FUNCTION_BLOCK PUBLIC PAEEMotor2D2P EXTENDS PAEEMotorStartCtrl
VAR_INPUT
END_VAR
VAR_OUTPUT
END_VAR
VAR
	_PAPointMatInOut1 : PAPoint(THIS^);
	_PAPointMatInOut2 : PAPoint(THIS^);
	_DirectionLeft : BOOL;
	_ReqDirectionLeft : BOOL;
	_ReqSpeedFast : BOOL;
	_SpeedFast : BOOL;
	_ToggleAllowed : BOOL;
	_TransitTimeSlowFast : TIME;
END_VAR

{attribute 'monitoring' := 'call'}
//{attribute 'TcRpcEnable'}
PROPERTY PUBLIC DirectionLeft : BOOL
GET // PUBLIC
DirectionLeft := _DirectionLeft;
END_GET
SET
_DirectionLeft := DirectionLeft;
Root.OnPropertyChangedBool(THIS^, 51, _DirectionLeft);
END_SET
END_PROPERTY

METHOD FB_init : BOOL
VAR_INPUT
	bInitRetains : BOOL; // if TRUE, the retain variables are initialized (warm start / cold start)
	bInCopyCode : BOOL;  // if TRUE, the instance afterwards gets moved into the copy code (online change)
	parent : IACComponent;
END_VAR
AddPoint(_PAPointMatInOut1);
AddPoint(_PAPointMatInOut2);
END_METHOD

METHOD FB_postinit
VAR_INPUT
	root : IACVariobatch;	
END_VAR
SUPER^.FB_postinit(root);  
root.OnPropertyChangedTime(THIS^, 50, _TransitTimeSlowFast);
root.OnPropertyChangedBool(THIS^, 51, _DirectionLeft);
root.OnPropertyChangedBool(THIS^, 52, _SpeedFast);
root.OnPropertyChangedBool(THIS^, 53, _ReqDirectionLeft);
root.OnPropertyChangedBool(THIS^, 54, _ReqSpeedFast);
END_METHOD

METHOD PUBLIC HasPointReachedOffPosition : BOOL
VAR_INPUT
	point : IACPoint;
END_VAR
IF point = PAPointMatInOut1 OR point = PAPointMatInOut2 THEN
	HasPointReachedOffPosition := NOT _RunState;
ELSE
	HasPointReachedOffPosition := FALSE;
END_IF
END_METHOD

METHOD PUBLIC HasPointReachedOnPosition : BOOL
VAR_INPUT
	point : IACPoint;
END_VAR
IF point = PAPointMatInOut1 THEN
	HasPointReachedOnPosition :=	( 	(NOT _DirectionLeft) 
									 AND _RunState 
									 AND (   (_ReqSpeedFast AND _SpeedFast) 
									 	  OR (NOT _ReqSpeedFast AND NOT _SpeedFast))
									)
								OR _DirectionLeft; // Fungiert als Eingangspunkt
ELSIF point = PAPointMatInOut2 THEN
	HasPointReachedOnPosition := 	(	_DirectionLeft 
									AND _RunState 
									AND (   (_ReqSpeedFast AND _SpeedFast) 
									 	 OR (NOT _ReqSpeedFast AND NOT _SpeedFast))
									)
								OR NOT _DirectionLeft; // Fungiert als Eingangspunkt
ELSE
	HasPointReachedOnPosition := FALSE;
END_IF
END_METHOD

METHOD PUBLIC InvokeSetterBool
VAR_INPUT
	PropertyID : INT;
	PropertyValue : BOOL;
END_VAR
SUPER^.InvokeSetterBool(PropertyID, PropertyValue);
IF PropertyID = 51 THEN
	DirectionLeft := PropertyValue;
ELSIF PropertyID = 52 THEN	
	SpeedFast := PropertyValue;
ELSIF PropertyID = 53 THEN	
	ReqDirectionLeft := PropertyValue;
ELSIF PropertyID = 54 THEN	
	ReqSpeedFast := PropertyValue;
END_IF
END_METHOD

METHOD PUBLIC InvokeSetterTime
VAR_INPUT
	PropertyID : INT;
	PropertyValue : DINT;
END_VAR
SUPER^.InvokeSetterTime(PropertyID, PropertyValue);
CASE PropertyID OF
	50:
		TransitTimeSlowFast := TO_TIME(PropertyValue);
END_CASE
END_METHOD

METHOD PUBLIC IsEnabledTurnOnFastLeft : BOOL
VAR_INPUT
END_VAR
END_METHOD

METHOD PUBLIC IsEnabledTurnOnFastRight : BOOL
VAR_INPUT
END_VAR
END_METHOD

METHOD PUBLIC IsEnabledTurnOnSlowLeft : BOOL
VAR_INPUT
END_VAR
END_METHOD

METHOD PUBLIC IsEnabledTurnOnSlowRight : BOOL
VAR_INPUT
END_VAR
END_METHOD

METHOD OnInitMemory
VAR_INPUT
	root : IACVariobatch;
END_VAR
RegisterProperty(root, 50, GCL.cSizeTIME); //TransitTimeSlowFast
RegisterProperty(root, 51, GCL.cSizeBYTE); //DirectionLeft
RegisterProperty(root, 52, GCL.cSizeBYTE); //SpeedFast
RegisterProperty(root, 53, GCL.cSizeBYTE); //ReqDirectionLeft
RegisterProperty(root, 54, GCL.cSizeBYTE); //ReqSpeedFast
SUPER^.OnInitMemory(root);
END_METHOD

PROPERTY PUBLIC PAPointMatInOut1 : IACPoint
GET
PAPointMatInOut1 := _PAPointMatInOut1;
END_GET
END_PROPERTY

PROPERTY PUBLIC PAPointMatInOut2 : IACPoint
GET // PUBLIC
PAPointMatInOut2 := _PAPointMatInOut2;
END_GET
END_PROPERTY

{attribute 'monitoring' := 'call'}
//{attribute 'TcRpcEnable'}
PROPERTY PUBLIC ReqDirectionLeft : BOOL
GET // PUBLIC
ReqDirectionLeft := _ReqDirectionLeft;
END_GET
SET // PUBLIC
_ReqDirectionLeft := ReqDirectionLeft;
Root.OnPropertyChangedBool(THIS^, 53, _ReqDirectionLeft);
IF Root.InSimulation THEN
	DirectionLeft := _ReqDirectionLeft;
END_IF
END_SET
END_PROPERTY

{attribute 'monitoring' := 'call'}
//{attribute 'TcRpcEnable'}
PROPERTY PUBLIC ReqSpeedFast : BOOL
GET // PUBLIC
ReqSpeedFast := _ReqSpeedFast;
END_GET
SET // PUBLIC
_ReqSpeedFast := ReqSpeedFast;
Root.OnPropertyChangedBool(THIS^, 54, _ReqSpeedFast);
IF Root.InSimulation THEN
	SpeedFast := _ReqSpeedFast;
END_IF
END_SET
END_PROPERTY

{attribute 'monitoring' := 'call'}
//{attribute 'TcRpcEnable'}
PROPERTY PUBLIC SpeedFast : BOOL
GET
SpeedFast := _SpeedFast;
END_GET
SET // PUBLIC
_SpeedFast := SpeedFast;
Root.OnPropertyChangedBool(THIS^, 52, _SpeedFast);
END_SET
END_PROPERTY

{attribute 'monitoring' := 'call'}
//{attribute 'TcRpcEnable'}
PROPERTY PUBLIC ToggleAllowed : BOOL
GET // PUBLIC
ToggleAllowed := _ToggleAllowed;
END_GET
SET // PUBLIC
_ToggleAllowed := ToggleAllowed;
END_SET
END_PROPERTY

{attribute 'monitoring' := 'call'}
//{attribute 'TcRpcEnable'}
PROPERTY PUBLIC TransitTimeSlowFast : TIME
GET // PUBLIC
TransitTimeSlowFast := _TransitTimeSlowFast;
END_GET
SET // PUBLIC
_TransitTimeSlowFast := TransitTimeSlowFast;
Root.OnPropertyChangedTime(THIS^, 50, _TransitTimeSlowFast);
END_SET
END_PROPERTY

METHOD PUBLIC TurnOnFastLeft
VAR_INPUT
END_VAR
END_METHOD

METHOD PUBLIC TurnOnFastRight
VAR_INPUT
END_VAR
END_METHOD

METHOD PUBLIC TurnOnSlowLeft
VAR_INPUT
END_VAR
END_METHOD

METHOD PUBLIC TurnOnSlowRight
VAR_INPUT
END_VAR
END_METHOD

END_FUNCTION_BLOCK

(* stored: Version 1.1.0.1, ProductVersion 3.1.4024.6
   POU PAEEMotor2D2P: Id {3f5f740c-9bfd-48df-8955-a3dfd86476a7}, SpecialFunc None
   Property DirectionLeft: Id {ed3ff90f-bcc4-49c9-8761-31d9d9624016}
   Get Get: Id {f6dc5d98-06b6-432e-af7d-35a3a0fd72b4}
   Set Set: Id {3edb5c4d-1f99-4b28-9d7d-f33340e0ddd3}
   Method FB_init: Id {cb962b15-023e-4e9c-bde3-fbf834738e9a}
   Method FB_postinit: Id {de3f108b-b7f2-451e-a281-50b9e0cdc5f0}
   Method HasPointReachedOffPosition: Id {52500e5a-2cbd-4e31-95d7-fb4c24a154bb}
   Method HasPointReachedOnPosition: Id {775d5d48-7abd-4846-96c7-21d5d986ae40}
   Method InvokeSetterBool: Id {1b7fc5d0-c5f2-4e80-a927-97f36ad5883d}
   Method InvokeSetterTime: Id {ea275111-c7e4-49e4-b253-36f38a4b74bc}
   Method IsEnabledTurnOnFastLeft: Id {095620b2-e94e-426b-9adc-e80da2c2d9f2}
   Method IsEnabledTurnOnFastRight: Id {025ef2ad-a140-44e5-9218-7f52ae579e12}
   Method IsEnabledTurnOnSlowLeft: Id {a0e7d9c2-a2c8-47a3-bdc0-759b189e0a72}
   Method IsEnabledTurnOnSlowRight: Id {ecaeb439-942e-4d04-b9dd-2b2c3487e92a}
   Method OnInitMemory: Id {5fff14d6-ea95-4167-bbf5-7a774d35e837}
   Property PAPointMatInOut1: Id {ce7eb083-070c-471e-83be-a65d1c841d31}
   Get Get: Id {84720b4d-238f-4f29-885c-02ab119f4746}
   Property PAPointMatInOut2: Id {82e7fbc2-3970-4c49-bcc2-23609c2bc019}
   Get Get: Id {59a55cd7-fab3-4af3-89e0-140f3502ca7e}
   Property ReqDirectionLeft: Id {b0d4afd9-8d0a-4f87-8f81-022a9274185d}
   Get Get: Id {ce9f8243-e14b-47b8-8cf1-011d5b167c94}
   Set Set: Id {d7b27653-3c4c-488b-acfe-c39f9144f5f0}
   Property ReqSpeedFast: Id {187177d4-ea49-4da7-90f5-61a0bf748802}
   Get Get: Id {ecfdc6cd-9972-42ee-8da5-0c36730ca586}
   Set Set: Id {9eb43bfa-0f45-4c81-9846-986ae543bb56}
   Property SpeedFast: Id {04fa51ea-deab-480c-80eb-5bd5933b5783}
   Get Get: Id {3800fea8-9749-496d-9741-f57484383f3d}
   Set Set: Id {bcd7bca2-8a8e-431f-be6d-2c4a5419080b}
   Property ToggleAllowed: Id {f08ee637-0898-4e5f-a72c-96600adefe18}
   Get Get: Id {b1f5e305-fa5c-4096-b908-6dc21694ea1f}
   Set Set: Id {e2f8682f-a55e-445e-92b5-84eca479b338}
   Property TransitTimeSlowFast: Id {9aa6f619-7d04-4ac2-bfdf-53695149b91b}
   Get Get: Id {c9f57aa8-2420-4c2b-b64b-99cedcb6d5d3}
   Set Set: Id {510af53e-7e85-41cd-95b1-0485e25c13f2}
   Method TurnOnFastLeft: Id {01147020-63e3-40b2-a9bd-8b368b487cb7}
   Method TurnOnFastRight: Id {5cd8d378-3f4c-42f1-a07d-172c1a072ffd}
   Method TurnOnSlowLeft: Id {d9290f2b-d40e-4759-a23b-32c1d8ae8652}
   Method TurnOnSlowRight: Id {62d3a9dd-9d83-4f21-840d-03e9f093b89e} *)
